// TIA Portal V19 export
TYPE "C301_STU_CLUST_TYPIC"
   STRUCT
      CMD_CAPA_CAPA { ExternalAccessible := 'False'; ExternalVisible := 'False'; ExternalWritable := 'False'} : USInt;   // Sturing ventilatie algemeen
      CMD_DIR { ExternalAccessible := 'False'; ExternalVisible := 'False'; ExternalWritable := 'False'} : USInt;   // Sturing richting
      CMD_ONHD { ExternalAccessible := 'False'; ExternalVisible := 'False'; ExternalWritable := 'False'} : USInt;   // Cluster die automatische onderhoudstesten moet uitvoeren
      VGV_BEV { ExternalAccessible := 'False'; ExternalVisible := 'False'; ExternalWritable := 'False'} : USInt;   // Vrijgave ventilator-beveiligingen onbalans en temperatuur
   END_STRUCT;
END_TYPE
